FUNCTION_BLOCK F_MUL_3 (* Multiplies three values *)
  (* Standard: 61131-3; Classification: standard arithmetic function; Description: Copyright (c) 2011, 2026 TU Wien ACIN, Patrick Aigner, HR Agrartechnik GmbH This program and the accompanying materials are made available under the terms of the Eclipse Public License 2.0 which is available at https://www.eclipse.org/legal/epl-2.0/ SPDX-License-Identifier: EPL-2.0 Some portions generated by Gemini CLI *)
  (* Version 1.0, 2026-02-01, Franz Höpfinger, HR Agrartechnik GmbH, Copy over from F_MUL and made this Block *)
  PACKAGE iec61131::arithmetic;
  {SET_ATTRIBUTE(eclipse4diac::core::GenericClassName, 'GEN_MUL')}
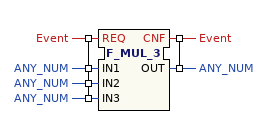
  EVENT_INPUT
    REQ WITH IN1, IN2, IN3; (* Normal Execution Request *)
  END_EVENT
  EVENT_OUTPUT
    CNF WITH OUT; (* Execution Confirmation *)
  END_EVENT
  VAR_INPUT
    IN1 : ANY_NUM; (* First function input *)
    IN2 : ANY_NUM; (* Second function input *)
    IN3 : ANY_NUM; (* Third function input *)
  END_VAR
  VAR_OUTPUT
    OUT : ANY_NUM; (* Result *)
  END_VAR
END_FUNCTION_BLOCK
